// TIA Portal V20 export
DATA_BLOCK "TorqueFB_TEL750_DB"   // DB45
// stored: InstanceOfName TorqueFB_TEL750, InstanceOfType FB
"TorqueFB_TEL750"
   // VAR_INPUT
   //    enable : Bool;
   //    refTorque : Real;
   //    addTorque : Real;
   //    upperLimit : Real;
   //    lowerLimit : Real;
   //    HWIDSTW : HW_IO;
   //    HWIDZSW : HW_IO;
   // END_VAR
   // VAR_OUTPUT
   //    busy : Bool;
   //    inUpperLimit : Bool;
   //    inLowerLimit : Bool;
   //    actTorque : Real;
   //    error : Bool;
   //    errorID : Word;
   //    diaID : Word;
   // END_VAR
   // VAR
   //    swSend : Array[0..2] of Word;
   //    swReceive : Word;
   //    sxSend : Struct
   //       M_ADD1 : Word;
   //       M_LIMIT_POS : Word;
   //       M_LIMIT_NEG : Word;
   //    END_STRUCT;
   //    sxReceive : Struct
   //       M_ACT : Word;
   //    END_STRUCT;
   // END_VAR
BEGIN
END_DATA_BLOCK
